{attribute 'qualified_only'}
{attribute 'strict'}
TYPE eInspectorResult : (
    NoAction := 0,
    Running := 10,
    Passed := 20,
    Failed := 30,
    Inconclusive := 35,
    Excluded := 40,
    Bypassed := 50
);
END_TYPE

(* stored: Version 1.1.0.1, ProductVersion 3.1.4024.9
   DUT eInspectorResult: Id {0144af4b-8ed9-0285-0c54-d5d7e851b8e5} *)
